TYPE ST_TempSave :
STRUCT
	stTempCmd							: ST_TempSave_Cmd;
END_STRUCT
END_TYPE

(* stored: Version 1.1.0.1, ProductVersion 3.1.4024.12
   DUT ST_TempSave: Id {444eec19-39db-48bc-8835-ef310eac201d} *)
